{attribute 'GeneratedUsingTerminal: EP4314-1002-0016'}
{attribute addProperty BoxType "EP4314-1002-0016"}
{attribute addProperty Id "InputAT %I*ARRAY[0..1] OF BOOL2TxPDO_StateAT %I*BOOL1TxPDO_ToggleAT %I*BOOL1"}
{attribute addProperty CRC "2573189997"}
{attribute addProperty Size "4"}
TYPE DI_Inputs_1F3A9325 EXTENDS InputBase_8311D824 :
STRUCT
	{attribute addProperty Name "Input"}
	Input AT %I* : ARRAY[0..1] OF BOOL;
	{attribute addProperty Name "TxPDO_State"}
	TxPDO_State AT %I* : BOOL;
	{attribute addProperty Name "TxPDO_Toggle"}
	TxPDO_Toggle AT %I* : BOOL;
END_STRUCT
END_TYPE

(* stored: Version 1.2.0.0, ProductVersion 3.1.4024.11
   DUT DI_Inputs_1F3A9325: Id {dc70a66d-9453-4af7-9495-b18d8e6e99c3} *)
